// Mitsubishi GX Works2 project: z10   PLC: Q02/Q02H

PROGRAM MAIN
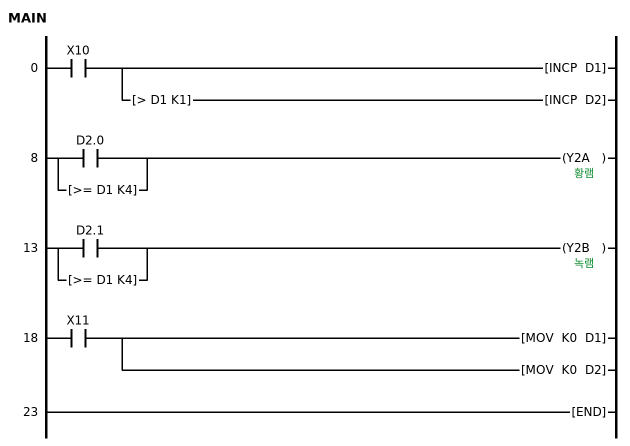
0     LD      X10
      INCP    D1
      AND>    D1 K1
      INCP    D2
8     LD      D2.0
      OR>=    D1 K4
      OUT     Y2A  ; 황램
13    LD      D2.1
      OR>=    D1 K4
      OUT     Y2B  ; 녹램
18    LD      X11
      MOV     K0 D1
      MOV     K0 D2
23    END
END_PROGRAM

// device comments not shown above
X0  ; 공급_후
X1  ; 공급_전
X2  ; 드릴_상
X3  ; 드릴_하
X4  ; 송출_후
X5  ; 송출_전
X6  ; 배출_후
X7  ; 배출_전
X8  ; 매거진
X9  ; 이송감지
X0A  ; 비금속
X0B  ; 금속
X0C  ; PB1
X0D  ; PB2
X0E  ; PB3
X0F  ; 비상정지
Y20  ; 공급_전
Y21  ; 공급_후
Y22  ; 드릴_실
Y23  ; 송출_전
Y24  ; 송출_후
Y25  ; 배출_전
Y26  ; 배출_후
Y27  ; 드릴_모
Y28  ; 컨베
Y29  ; 적램
